{attribute 'enable_dynamic_creation'}
FUNCTION_BLOCK EtherCATDevice IMPLEMENTS I_EtherCATDevice
VAR_INPUT
END_VAR
VAR_OUTPUT
END_VAR
VAR
END_VAR

METHOD IsDeviceOK : BOOL
VAR_INPUT
END_VAR
END_METHOD

END_FUNCTION_BLOCK

(* stored: Version 1.1.0.1, ProductVersion 3.1.4024.12
   POU EtherCATDevice: Id {af8f1906-b637-4799-829a-dc8018136702}, SpecialFunc None
   Method IsDeviceOK: Id {bfa56fa0-7124-4f0f-b373-cf9908c856da} *)
